// TIA Portal V17 export
// export: Created 2021-09-08T12:46:16.1780561Z, ExportSetting WithDefaults, DisplayName Totally Integrated Automation Portal, DisplayVersion V17, DisplayName TIA Portal Openness, DisplayVersion V17, DisplayName TIA Portal Version Control Interface, DisplayVersion V17, DisplayName STEP 7 Professional, DisplayVersion V17, DisplayName STEP 7 Safety, DisplayVersion V17, DisplayName WinCC Advanced, DisplayVersion V17
TYPE "FREQ_COUNTER"
// stored: IsFailsafeCompliant false
   STRUCT
      litrsPerPuls : UInt;
      prewHour : UInt;
      curHour : UInt;
      prewDay : UDInt;
      curDay : UDInt;
      all : UDInt;
      rst : Bool;
   END_STRUCT;
END_TYPE
